{attribute 'qualified_only'}
{attribute 'strict'}
TYPE eConditionCheck :
(
	enum_member := 0
);
END_TYPE

(* stored: Version 1.1.0.1, ProductVersion 3.1.4024.12
   DUT eConditionCheck: Id {a286c164-0e4a-4060-8654-dbb16d2c3ee8} *)
